Fanuc KAREL source: INI_DYN_DISB.kl

PROGRAM T
%NOLOCKGROUP
VAR
 v0 : BOOLEAN
 v1 : STRING[40]
 v2 : INTEGER
 v3 : INTEGER
 v4 : INTEGER
 v5 : INTEGER
 v6 : INTEGER
 v7 : INTEGER
 v8 : ARRAY[10] OF STRING[40]
 v9 : INTEGER
BEGIN
 INI_DYN_DISB(v0, v1, v2, v3, v4, v5, v6, v7, v8, v9)
END T
